% RSLogix 500 project INTRO TO PLC - JOB 16.RSS, saved by version 10.00.00.00 %
PROJECT "PL06B"    % processor: Bul.1763 MicroLogix 1100 Series B %

PROGRAM FILES
  LAD 2   8 rungs

DATA FILES
  O0 OUTPUT  4 elements
  I1 INPUT  6 elements
  S2 STATUS  66 elements
  B3 BINARY  1 elements
  T4 TIMER  2 elements
  C5 COUNTER  2 elements
  R6 CONTROL  1 elements
  N7 INTEGER  1 elements
  F8 FLOAT  1 elements

LADDER 2
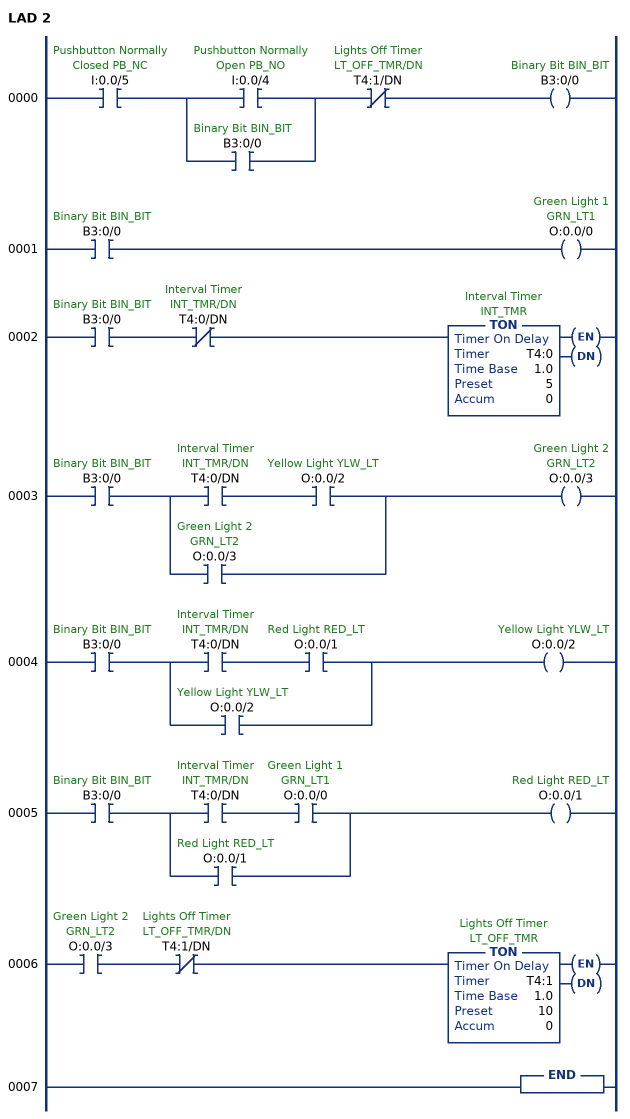
% Rung: 0 %
SOR XIC I:0.0/5 BST XIC I:0.0/4 NXB XIC B3:0/0 BND XIO T4:1/DN OTE B3:0/0 EOR
%   I:0.0/5  PB_NC  "Pushbutton Normally Closed" %
%   I:0.0/4  PB_NO  "Pushbutton Normally Open" %
%   B3:0/0  BIN_BIT  "Binary Bit" %
%   T4:1  LT_OFF_TMR  "Lights Off Timer" %
% Rung: 1 %
SOR XIC B3:0/0 OTE O:0.0/0 EOR
%   B3:0/0  BIN_BIT  "Binary Bit" %
%   O:0.0/0  GRN_LT1  "Green Light 1" %
% Rung: 2 %
SOR XIC B3:0/0 XIO T4:0/DN TON T4:0 1.0 5 0 EOR
%   B3:0/0  BIN_BIT  "Binary Bit" %
%   T4:0  INT_TMR  "Interval Timer" %
% Rung: 3 %
SOR XIC B3:0/0 BST XIC T4:0/DN XIC O:0.0/2 NXB XIC O:0.0/3 BND OTE O:0.0/3 EOR
%   B3:0/0  BIN_BIT  "Binary Bit" %
%   T4:0  INT_TMR  "Interval Timer" %
%   O:0.0/2  YLW_LT  "Yellow Light" %
%   O:0.0/3  GRN_LT2  "Green Light 2" %
% Rung: 4 %
SOR XIC B3:0/0 BST XIC T4:0/DN XIC O:0.0/1 NXB XIC O:0.0/2 BND OTE O:0.0/2 EOR
%   B3:0/0  BIN_BIT  "Binary Bit" %
%   T4:0  INT_TMR  "Interval Timer" %
%   O:0.0/1  RED_LT  "Red Light" %
%   O:0.0/2  YLW_LT  "Yellow Light" %
% Rung: 5 %
SOR XIC B3:0/0 BST XIC T4:0/DN XIC O:0.0/0 NXB XIC O:0.0/1 BND OTE O:0.0/1 EOR
%   B3:0/0  BIN_BIT  "Binary Bit" %
%   T4:0  INT_TMR  "Interval Timer" %
%   O:0.0/0  GRN_LT1  "Green Light 1" %
%   O:0.0/1  RED_LT  "Red Light" %
% Rung: 6 %
SOR XIC O:0.0/3 XIO T4:1/DN TON T4:1 1.0 10 0 EOR
%   O:0.0/3  GRN_LT2  "Green Light 2" %
%   T4:1  LT_OFF_TMR  "Lights Off Timer" %
% Rung: 7 %
SOR END EOR

OTHER DOCUMENTED ADDRESSES
  B3:0/1  SEAL2  "Seal 2"
  C5:0  CYC_CTR  "Cycle Counter"
  C5:1  CYC_CTR2  "Cycle Counter 2"
  I:0.0/0  SS1A  "Selector Switch 1 Position A"
  I:0.0/1  SS1B  "Selector Switch 1 Position B"
  I:0.0/2  SS2A  "Selector Switch 2 Position A"
  I:0.0/3  SS2B  "Selector Switch 2 Position B"

DATA TABLE (non-zero values as saved)
DATA T4
% .PRE .ACC %
% T4:0 % 5 0
% T4:1 % 10 0
DATA C5
% .PRE .ACC %
% C5:0 % 30 0
% C5:1 % 5 5
